Staubli VAL3: onEditItem.pgx

public program onEditItem(string& x_sEvent[], num x_nIndex, num x_nIndexItem)
begin
  if x_nIndex!=6
    // edit the custom element that was add in the list
    call onEditTrsf(x_nIndex,x_nIndexItem,x_sEvent)
  elseIf x_nIndex==6
    call changePCircle(x_nIndexItem)
  endIf
end
